// TIA Portal V18 export
DATA_BLOCK "SireneMain_DB"   // DB10
VERSION : 0.1
// stored: AutoNumber true, DBAccessibleFromOPCUA true, DBAccessibleFromWebserver true, InstanceOfName SireneMain, InstanceOfType FB
"SireneMain"
   // VAR
   //    sirene_Instance { S7_SetPoint := 'True'} : "sirene_v2";
   // END_VAR
BEGIN
END_DATA_BLOCK
